Xinje XDPPro project, PLC1: XD5-48T6 (software 3.7.4b 2021-06-17)

PROGRAM Ladder

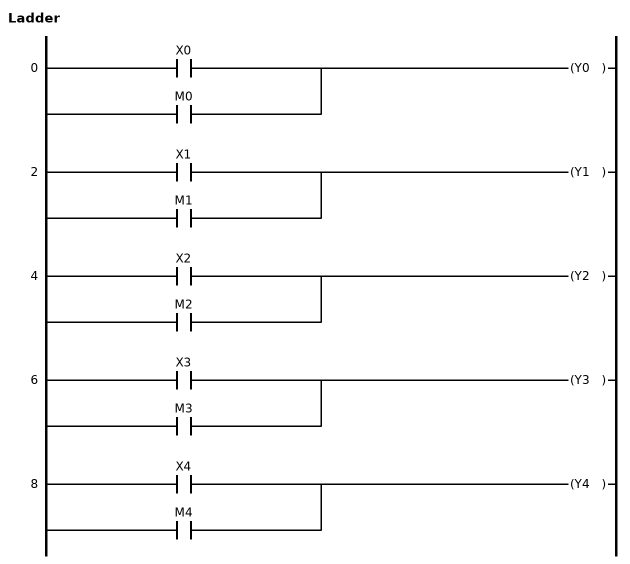
LD     X0
OR     M0
OUT    Y0
LD     X1
OR     M1
OUT    Y1
LD     X2
OR     M2
OUT    Y2
LD     X3
OR     M3
OUT    Y3
LD     X4
OR     M4
OUT    Y4